// TwinCAT 3 PLC project UdpComm
// ProgramVersion: 3.1.4020.10
// libraries:
//   Tc2_Standard, * (Beckhoff Automation GmbH)
//   Tc2_System, * (Beckhoff Automation GmbH)
//   Tc2_Utilities, * (Beckhoff Automation GmbH)
//   Tc3_Interfaces, * (Beckhoff Automation GmbH)
//   Tc3_Module, * (Beckhoff Automation GmbH)
// project tree:
//   DUTs/ ModeStewart.TcDUT, RxRemote.TcDUT, ControlComau.TcDUT, RxComau.TcDUT, TxComau.TcDUT, RxMru.TcDUT, ControlStewart.TcDUT, TxRemote.TcDUT, FeedbackLeica.TcDUT, FeedbackComau.TcDUT, FeedbackMru.TcDUT, FeedbackStewart.TcDUT, TxHmi.TcDUT, TxHmiComau.TcDUT, TxHmiLeica.TcDUT, TxHmiMru.TcDUT, TxHmiStewart.TcDUT, TxStewart.TcDUT, RxStewart.TcDUT
//   / GlobalTextList.TcGTLO, TaskMAIN.TcTTO, Visualization Manager.TcVMO (not stored)
//   POUs/Kinematics/ EulerToBody.TcPOU, StewartTransform.TcPOU, xyz2zyx.TcPOU, zyx2xyz.TcPOU
//   POUs/LabEquipment/ LeicaInterface.TcPOU, RemoteInterface.TcPOU, MruInterface.TcPOU, ComauInterface.TcPOU, StewartInterface.TcPOU
//   POUs/ MAIN.TcPOU
//   POUs/Ship Simulation/ ShipSimulator.TcPOU, StocWave.TcPOU
//   POUs/UdpFBs/ FB_UdpClient.TcPOU (not stored), FB_UdpServer.TcPOU
// real-time tasks:
//   TASK TaskMAIN: cycle T#5ms, priority 20, ADS port 350
// I/O:
//   DEVICE EM1500 (RT-Ethernet Adapter)
//   DEVICE EM8000 (RT-Ethernet Adapter)
//   DEVICE COMAU (RT-Ethernet Adapter)
//   DEVICE REMOTE (RT-Ethernet Adapter)
//   DEVICE MRU2 (RT-Ethernet Adapter)
//   DEVICE MRU1 (RT-Ethernet Adapter)
//   DEVICE LeicaAT960 (EtherCAT), AmsNetId 169.254.76.98.11.1
//     Box 1 (Leica-RT-Output) [Leica RT Output]
// variable links:
//   UdpComm/UdpComm Instance <-> LeicaAT960 (EtherCAT)/Box 1 (Leica-RT-Output)
//     TaskMAIN Inputs/MAIN.at960.AngleHz <-> Cyclic Measurements/AngleHz
//     TaskMAIN Inputs/MAIN.at960.AngleVt <-> Cyclic Measurements/AngleVt
//     TaskMAIN Inputs/MAIN.at960.Distance <-> Cyclic Measurements/Distance
//     TaskMAIN Inputs/MAIN.at960.Quaternion{0..3} <-> Cyclic Measurements/Quaternion{0..3}  (4 links)
//     TaskMAIN Inputs/MAIN.at960.TimeStamp <-> Cyclic Measurements/TimeStamp

CONFIGURATION UdpComm
    RESOURCE PLC ON TwinCAT3
        TASK TaskMAIN(INTERVAL := T#5ms, PRIORITY := 20);
        PROGRAM MAIN WITH TaskMAIN : MAIN;
    END_RESOURCE
END_CONFIGURATION

// ---- DUTs/ModeStewart.TcDUT

TYPE ModeStewart :
(
	MODE_IDLE := 0,
	MODE_SIMULATOR,
	MODE_REMOTE,
	MODE_TRANSITION,
	MODE_GENERATOR,
	MODE_STOP
);
END_TYPE

// ---- DUTs/RxRemote.TcDUT
TYPE RxRemote :
STRUCT
	udp_key : DINT;
	comau : ControlComau;
END_STRUCT
END_TYPE

// ---- DUTs/ControlComau.TcDUT
TYPE ControlComau :
STRUCT
	q1 : REAL;
	q2 : REAL;
	q3 : REAL;
	q4 : REAL;
	q5 : REAL;
	q6 : REAL;
	q1_t : REAL;
	q2_t : REAL;
	q3_t : REAL;
	q4_t : REAL;
	q5_t : REAL;
	q6_t : REAL;
	q1_tt : REAL;
	q2_tt : REAL;
	q3_tt : REAL;
	q4_tt : REAL;
	q5_tt : REAL;
	q6_tt : REAL;
END_STRUCT
END_TYPE

// ---- DUTs/RxComau.TcDUT
TYPE RxComau :
STRUCT
	modalityActive : DINT;
	q1_ref : REAL;
	q2_ref : REAL;
	q3_ref : REAL;
	q4_ref : REAL;
	q5_ref : REAL; 
	q6_ref : REAL;
	q1 : REAL;
	q2 : REAL;
	q3 : REAL;
	q4 : REAL;
	q5 : REAL; 
	q6 : REAL;
	q1_t : REAL;
	q2_t : REAL;
	q3_t : REAL;
	q4_t : REAL;
	q5_t : REAL;
	q6_t : REAL;
	q1_tt : REAL;
	q2_tt : REAL;
	q3_tt : REAL;
	q4_tt : REAL;
	q5_tt : REAL;
	q6_tt : REAL;
END_STRUCT
END_TYPE

// ---- DUTs/TxComau.TcDUT
TYPE TxComau :
STRUCT
	udp_key	: DINT := 0;
	cmnd : DINT := 0;
	omega : REAL := 1.0;
	beta : REAL := 1.0;
	q1 : REAL := 0.0;
	q2 : REAL := 0.0;
	q3 : REAL := -90.0;
	q4 : REAL := 0.0;
	q5 : REAL := 90.0;
	q6 : REAL := 0.0;
	q1_t : REAL := 0.0;
	q2_t : REAL := 0.0;
	q3_t : REAL := 0.0;
	q4_t : REAL := 0.0;
	q5_t : REAL := 0.0;
	q6_t : REAL := 0.0;
	q1_tt : REAL := 0.0;
	q2_tt : REAL := 0.0;
	q3_tt : REAL := 0.0;
	q4_tt : REAL := 0.0;
	q5_tt : REAL := 0.0;
	q6_tt : REAL := 0.0;
END_STRUCT
END_TYPE

// ---- DUTs/RxMru.TcDUT
{attribute 'pack_mode' := '1'}
TYPE RxMru :
STRUCT
	mruOK : BYTE;
	dataLength : BYTE;
	token : BYTE;
	Temperature : REAL;
	PosMru_D : REAL;
	VelMru_D : REAL;
	AccMru_D : REAL;
	AngRate_D : REAL;
	Roll : REAL;
	Pitch : REAL;
	Yaw	: REAL;
	AngRate_R : REAL;
	AngRate_P : REAL;
	AngRate_Y : REAL;
	AngAcc_R : REAL;
	AngAcc_P : REAL;
	AngAcc_Y : REAL;
	VelMru_R : REAL;
	VelMru_P : REAL;
	VelMru_Y : REAL;
	AccMru_R : REAL;
	AccMru_P : REAL;
	AccMru_Y : REAL;
	checksum : BYTE;
END_STRUCT
END_TYPE

// ---- DUTs/ControlStewart.TcDUT
TYPE ControlStewart :
STRUCT
	surge : REAL := 0.0;
	sway : REAL := 0.0;
	heave : REAL := 0.0;
	phi : REAL := 0.0;
	theta : REAL := 0.0;
	psi : REAL := 0.0;
END_STRUCT
END_TYPE

// ---- DUTs/TxRemote.TcDUT
TYPE TxRemote :
STRUCT
	t : REAL := 0.0;
	em8000 : FeedbackStewart;	
	em1500 : FeedbackStewart;
	comau : FeedbackComau;
	at960 : FeedbackLeica;
	mru1 : FeedbackMru;
	mru2 : FeedbackMru;
END_STRUCT
END_TYPE

// ---- DUTs/FeedbackLeica.TcDUT
TYPE FeedbackLeica :
STRUCT
	x : REAL;
	y : REAL;
	z : REAL;
	q0 : REAL;
	q1 : REAL;
	q2 : REAL;
	q3 : REAL;
END_STRUCT
END_TYPE

// ---- DUTs/FeedbackComau.TcDUT
TYPE FeedbackComau :
STRUCT
	q1 : REAL;
	q2 : REAL;
	q3 : REAL;
	q4 : REAL;
	q5 : REAL;
	q6 : REAL;
	q1_t : REAL;
	q2_t : REAL;
	q3_t : REAL;
	q4_t : REAL;
	q5_t : REAL;
	q6_t : REAL;
	q1_tt : REAL;
	q2_tt : REAL;
	q3_tt : REAL;
	q4_tt : REAL;
	q5_tt : REAL;
	q6_tt : REAL;
END_STRUCT
END_TYPE

// ---- DUTs/FeedbackMru.TcDUT
TYPE FeedbackMru :
STRUCT
	heave : REAL;
	heave_t : REAL;
	heave_tt : REAL;
	turn_rate : REAL;
	roll : REAL;
	pitch : REAL;
	yaw : REAL;
	wx : REAL;
	wy : REAL;
	wz : REAL;
	wx_t : REAL;
	wy_t : REAL;
	wz_t : REAL;
	x_t : REAL;
	y_t : REAL;
	z_t : REAL;
	x_tt : REAL;
	y_tt : REAL;
	z_tt : REAL;
END_STRUCT
END_TYPE

// ---- DUTs/FeedbackStewart.TcDUT
TYPE FeedbackStewart :
STRUCT
	surge : REAL;
	sway : REAL;
	heave : REAL;
	phi : REAL;
	theta : REAL;
	psi	: REAL;
	surge_t	: REAL;
	sway_t	: REAL;
	heave_t	: REAL;
	wx : REAL;
	wy : REAL;
	wz : REAL;
	surge_tt : REAL;
	sway_tt : REAL;
	heave_tt : REAL;
	wx_t : REAL;
	wy_t : REAL;
	wz_t : REAL;
END_STRUCT
END_TYPE

// ---- DUTs/TxHmi.TcDUT
TYPE TxHmi :
STRUCT
	t : REAL := 0.0;
	em1500 : TxHmiStewart;
	em8000 : TxHmiStewart;
	comau : TxHmiComau;
	at960 : TxHmiLeica;	
	mru1 : TxHmiMru;
	mru2 : TxHmiMru;
END_STRUCT
END_TYPE

// ---- DUTs/TxHmiComau.TcDUT
TYPE TxHmiComau :
STRUCT
	status : DINT;
	q1 : REAL;
	q2 : REAL;
	q3 : REAL;
	q4 : REAL;
	q5 : REAL;
	q6 : REAL;
END_STRUCT
END_TYPE

// ---- DUTs/TxHmiLeica.TcDUT
TYPE TxHmiLeica :
STRUCT
	status : DINT;
	x : REAL;
	y : REAL;
	z : REAL;
	q0 : REAL;
	q1 : REAL;
	q2 : REAL;
	q3 : REAL;
END_STRUCT
END_TYPE

// ---- DUTs/TxHmiMru.TcDUT
TYPE TxHmiMru :
STRUCT
	status : DINT;
END_STRUCT
END_TYPE

// ---- DUTs/TxHmiStewart.TcDUT
TYPE TxHmiStewart :
STRUCT
	status : DINT;
	surge : REAL;
	sway : REAL;
	heave : REAL;
	phi : REAL;
	theta : REAL;
	psi	: REAL;
	surge_ref : REAL;
	sway_ref : REAL;
	heave_ref : REAL;
	phi_ref : REAL;
	theta_ref : REAL;
	psi_ref	: REAL;
	L1 : REAL;
	L2 : REAL;
	L3 : REAL;
	L4 : REAL;
	L5 : REAL;
	L6 : REAL;
	surge_sim : REAL;
	sway_sim : REAL;
	heave_sim : REAL;
	phi_sim : REAL;
	theta_sim : REAL;
	psi_sim	: REAL;
END_STRUCT
END_TYPE

// ---- DUTs/TxStewart.TcDUT
TYPE TxStewart :
STRUCT
	COUNT : DINT := 0;
	CMND : DINT := 0;
	AX : REAL := 0.0;
	AY : REAL := 0.0;
	AZ : REAL := 0.0;
	Dax : REAL := 0.0;
	Day : REAL := 0.0;
	Daz : REAL := 0.0;
	P_dot_CG : REAL := 0.0;
	Q_dot_CG : REAL := 0.0;
	R_dot_CG : REAL := 0.0;
	P_CG : REAL := 0.0;
	Q_CG : REAL := 0.0;
	R_CG : REAL := 0.0;
	Phi : REAL := 0.0;
	Theta : REAL := 0.0;
	U : REAL := 0.0;
	X_DIRECT : REAL := 0.0;
	Y_DIRECT : REAL := 0.0;
	Z_DIRECT : REAL := 0.0;
	X_CG : REAL := 0.0;
	Y_CG : REAL := 0.0;
	Z_CG : REAL := 0.0;
	Flags : REAL := 0.0;
	Bump_1 : REAL := 0.0;
	Bump_2 : REAL := 0.0;
	Bump_3 : REAL := 0.0;
	Bump_4 : REAL := 0.0;
	Bump_5 : REAL := 0.0;
	FREQ1 : REAL := 0.0;
	FREQ2 : REAL := 0.0;
	FREQ3 : REAL := 0.0;
	FREQ4 : REAL := 0.0;
	FREQ5 : REAL := 0.0;
	FREQ6 : REAL := 0.0;
	FREQ7 : REAL := 0.0;
	FREQ8 : REAL := 0.0;
	FREQ9 : REAL := 0.0;
	FREQ10 : REAL := 0.0;
	FREQ11 : REAL := 0.0;
	FREQ12 : REAL := 0.0;
	FREQ13 : REAL := 0.0;
	FREQ14 : REAL := 0.0;
	FREQ15 : REAL := 0.0;
	FREQ16 : REAL := 0.0;
	FREQ17 : REAL := 0.0;
	FREQ18 : REAL := 0.0;
	FREQ19 : REAL := 0.0;
	FREQ20 : REAL := 0.0;
	XGAIN1 : REAL := 0.0;
	XGAIN2 : REAL := 0.0;
	XGAIN3 : REAL := 0.0;
	XGAIN4 : REAL := 0.0;
	XGAIN5 : REAL := 0.0;
	XGAIN6 : REAL := 0.0;
	XGAIN7 : REAL := 0.0;
	XGAIN8 : REAL := 0.0;
	XGAIN9 : REAL := 0.0;
	XGAIN10 : REAL := 0.0;
	XGAIN11 : REAL := 0.0;
	XGAIN12 : REAL := 0.0;
	XGAIN13 : REAL := 0.0;
	XGAIN14 : REAL := 0.0;
	XGAIN15 : REAL := 0.0;
	XGAIN16 : REAL := 0.0;
	XGAIN17 : REAL := 0.0;
	XGAIN18 : REAL := 0.0;
	XGAIN19 : REAL := 0.0;
	XGAIN20 : REAL := 0.0;
	YGAIN1 : REAL := 0.0;
	YGAIN2 : REAL := 0.0;
	YGAIN3 : REAL := 0.0;
	YGAIN4 : REAL := 0.0;
	YGAIN5 : REAL := 0.0;
	YGAIN6 : REAL := 0.0;
	YGAIN7 : REAL := 0.0;
	YGAIN8 : REAL := 0.0;
	YGAIN9 : REAL := 0.0;
	YGAIN10 : REAL := 0.0;
	YGAIN11 : REAL := 0.0;
	YGAIN12 : REAL := 0.0;
	YGAIN13 : REAL := 0.0;
	YGAIN14 : REAL := 0.0;
	YGAIN15 : REAL := 0.0;
	YGAIN16 : REAL := 0.0;
	YGAIN17 : REAL := 0.0;
	YGAIN18 : REAL := 0.0;
	YGAIN19 : REAL := 0.0;
	YGAIN20 : REAL := 0.0;
	ZGAIN1 : REAL := 0.0;
	ZGAIN2 : REAL := 0.0;
	ZGAIN3 : REAL := 0.0;
	ZGAIN4 : REAL := 0.0;
	ZGAIN5 : REAL := 0.0;
	ZGAIN6 : REAL := 0.0;
	ZGAIN7 : REAL := 0.0;
	ZGAIN8 : REAL := 0.0;
	ZGAIN9 : REAL := 0.0;
	ZGAIN10 : REAL := 0.0;
	ZGAIN11 : REAL := 0.0;
	ZGAIN12 : REAL := 0.0;
	ZGAIN13 : REAL := 0.0;
	ZGAIN14 : REAL := 0.0;
	ZGAIN15 : REAL := 0.0;
	ZGAIN16 : REAL := 0.0;
	ZGAIN17 : REAL := 0.0;
	ZGAIN18 : REAL := 0.0;
	ZGAIN19 : REAL := 0.0;
	ZGAIN20 : REAL := 0.0;
	X_EXTRA : REAL := 0.0;
	Y_EXTRA : REAL := 0.0;
	Z_EXTRA : REAL := 0.0;
	PHI_EXTRA : REAL := 0.0;
	THETA_EXTRA : REAL := 0.0;
	PSI_EXTRA : REAL := 0.0;
	X_EXTRA_DOT : REAL := 0.0;
	Y_EXTRA_DOT : REAL := 0.0;
	Z_EXTRA_DOT : REAL := 0.0;
	PHI_EXTRA_DOT : REAL := 0.0;
	THETA_EXTRA_DOT : REAL := 0.0;
	PSI_EXTRA_DOT : REAL := 0.0;
	X_EXTRA_DDOT : REAL := 0.0;
	Y_EXTRA_DDOT : REAL := 0.0;
	Z_EXTRA_DDOT : REAL := 0.0;
	PHI_EXTRA_DDOT : REAL := 0.0;
	THETA_EXTRA_DDOT : REAL := 0.0;
	PSI_EXTRA_DDOT : REAL := 0.0;
END_STRUCT
END_TYPE

// ---- DUTs/RxStewart.TcDUT
TYPE RxStewart :
STRUCT
	Frame_Count : DINT := 0;
	Motion_Status : DINT := 0;
	Platform_setpoint_surge : REAL := 0.0;
	Platform_setpoint_sway : REAL := 0.0;
	Platform_setpoint_heave : REAL := 0.0;
	Platform_setpoint_roll : REAL := 0.0;
	Platform_setpoint_pitch : REAL := 0.0;
	Platform_setpoint_yaw : REAL := 0.0;
	Special_effect_surge_setpoint : REAL := 0.0;
	Special_effect_sway_setpoint : REAL := 0.0;
	Special_effect_heave_setpoint : REAL := 0.0;
	Special_effect_roll_setpoint : REAL := 0.0;
	Special_effect_pitch_setpoint : REAL := 0.0;
	Special_effect_yaw_setpoint : REAL := 0.0;
	Actual_position_actuator_1 : REAL := 0.0;
	Actual_position_actuator_2 : REAL := 0.0;
	Actual_position_actuator_3 : REAL := 0.0;
	Actual_position_actuator_4 : REAL := 0.0;
	Actual_position_actuator_5 : REAL := 0.0;
	Actual_position_actuator_6 : REAL := 0.0;
	Actual_platform_position_surge : REAL := 0.0;
	Actual_platform_position_sway : REAL := 0.0;
	Actual_platform_position_heave : REAL := 0.0;
	Actual_platform_position_roll : REAL := 0.0;
	Actual_platform_position_pitch : REAL := 0.0;
	Actual_platform_position_yaw : REAL := 0.0;
	Actual_platform_velocity_surge : REAL := 0.0;
	Actual_platform_velocity_sway : REAL := 0.0;
	Actual_platform_velocity_heave : REAL := 0.0;
	Actual_platform_velocity_roll : REAL := 0.0;
	Actual_platform_velocity_pitch : REAL := 0.0;
	Actual_platform_velocity_yaw : REAL := 0.0;
	Actual_platform_acceleration_surge : REAL := 0.0;
	Actual_platform_acceleration_sway : REAL := 0.0;
	Actual_platform_acceleration_heave : REAL := 0.0;
	Actual_platform_acceleration_roll : REAL := 0.0;
	Actual_platform_acceleration_pitch : REAL := 0.0;
	Actual_platform_acceleration_yaw : REAL := 0.0;
END_STRUCT
END_TYPE

// ---- POUs/MAIN.TcPOU
PROGRAM MAIN
VAR
	// HMI data
	hmi 				: TxHmi;	

	// Remote Interface	
	remote				: RemoteInterface(3232258620, 50060, 50050);
	
	// EtherCAT equipment
	at960				: LeicaInterface(ADR(hmi.at960));
	
	// UDP Equipment
	em1500				: StewartInterface(3232258591, 50031, 50041, 0, ADR(hmi.em1500));
	em8000				: StewartInterface(3232258590, 50030, 50040, 254, ADR(hmi.em8000));
	comau				: ComauInterface(3232258592, 50032, 50042, ADR(hmi.comau));
	
	mru1				: MruInterface(7551, ADR(hmi.mru1));
	mru2				: MruInterface(7552, ADR(hmi.mru2));
	
	
	counter				: UDINT := 0;
	
	
	
END_VAR

// Update remote data
remote();

// Update EtherCAT equipment
at960();

// Update UDP equipment
em1500();
em8000();
comau();
mru1();
mru2();

// Update timer
hmi.t := hmi.t + 5.0/1000.0;

END_PROGRAM

// ---- POUs/LabEquipment/RemoteInterface.TcPOU
{attribute 'c++_compatible'}
FUNCTION_BLOCK RemoteInterface IMPLEMENTS ITcIoUdpProtocolRecv
VAR_INPUT
	feedback			: TxRemote;
END_VAR
VAR_OUTPUT
	control 			: RxRemote;
END_VAR
VAR
	// UDP connection
	{attribute 'TcInitSymbol'}
	oid					: OTCID;
	ipUdp 				: ITcIoUdpProtocol;
	recvCounter			: UDINT := 0;
	sendCounter			: UDINT := 0;
	remoteUdpPort		: UINT;
	remoteIpAddr		: UDINT;	
	localUdpPort		: UINT;
	
	// UDP raw data
	rxUdpData			: RxRemote;
	txUdpData			: TxRemote;
	

END_VAR

VAR CONSTANT
	pi					: REAL := 3.141592653589793;
END_VAR


feedback.t := main.hmi.t;

// Update UDP data
UpdateUDP();

// Update IO data
UpdateIO();

METHOD FB_exit : BOOL
VAR_INPUT
	bInCopyCode : BOOL; // if TRUE, the exit method is called for exiting an instance that is copied afterwards (online change).
END_VAR
IF (NOT bInCopyCode AND ipUdp <> 0) THEN //Shutdown
	ipUdp.UnregisterReceiver(localUdpPort);
	FW_SafeRelease(ADR(ipUdp));
	FB_exit := TRUE;
ELSE
	FB_exit := FALSE;
END_IF
END_METHOD

METHOD FB_init : BOOL
VAR_INPUT
	bInitRetains 		: BOOL; // if TRUE, the retain variables are initialized (warm start / cold start)
	bInCopyCode 		: BOOL;  // if TRUE, the instance afterwards gets moved into the copy code (online change)
	
	_remoteIpAddr		: UDINT;
	_remoteUdpPort		: UINT;
	_localUdpPort		: UINT;
END_VAR

VAR
	ipSrv				: ITComObjectServer;
	hr 					: HRESULT;
END_VAR
// Initilize parameters
remoteIpAddr := _remoteIpAddr;
remoteUdpPort := _remoteUdpPort;
localUdpPort := _localUdpPort;

IF NOT bInCopyCode THEN // no online change
	IF ipUdp = 0 THEN
	    hr := FW_ObjMgr_GetObjectInstance(oid:=oid, iid:=TC_GLOBAL_IID_LIST.IID_ITcIoUdpProtocol, pipUnk:=ADR(ipUdp) );
		
		IF ( SUCCEEDED(hr) AND ipUdp.RegisterReceiver(localUdpPort, THIS^) = 0 ) THEN //open port
			FB_init := TRUE;
		ELSE
			FB_init := FALSE;			
			FW_SafeRelease(ADR(ipUdp));
		END_IF				
	END_IF
END_IF
END_METHOD

METHOD FB_reinit : BOOL
VAR_INPUT
END_VAR
IF (ipUdp <> 0) THEN 
  ipUdp.RegisterReceiver(localUdpPort, THIS^);
END_IF
END_METHOD

{attribute 'c++_compatible'}
{attribute 'signature_flag' := '33554688'}
{attribute 'pack_mode' := '4'}
{attribute 'show'}
{attribute 'minimal_input_size' := '4'}
{attribute 'checksuperglobal'}

METHOD ReceiveData : HRESULT
VAR_INPUT
	ipAddr	: UDINT;
	udpDestPort	: UINT;
	udpSrcPort	: UINT;
	nData	: UDINT;
	pData	: PVOID;
	pVlan	: POINTER TO ETYPE_VLAN_HEADER := 0;
END_VAR
IF (nData = SIZEOF(rxUdpData)) THEN
	// Copy recieved pData to rxUdpData
	MEMCPY(ADR(rxUdpData), pData, nData);
	
	// Count number of recieved UDP packets
	recvCounter := recvCounter + 1;
END_IF;
END_METHOD

{attribute 'c++_compatible'}
{attribute 'signature_flag' := '33554688'}
{attribute 'pack_mode' := '4'}
{attribute 'show'}
{attribute 'minimal_input_size' := '4'}
{attribute 'checksuperglobal'}

METHOD TcAddRef : UDINT
END_METHOD

{attribute 'c++_compatible'}
{attribute 'signature_flag' := '33554688'}
{attribute 'pack_mode' := '4'}
{attribute 'show'}
{attribute 'minimal_input_size' := '4'}
{attribute 'checksuperglobal'}

METHOD TcQueryInterface : HRESULT
VAR_INPUT
	iid	: REFERENCE TO IID;
	pipItf	: POINTER TO PVOID;
END_VAR
END_METHOD

{attribute 'c++_compatible'}
{attribute 'signature_flag' := '33554688'}
{attribute 'pack_mode' := '4'}
{attribute 'show'}
{attribute 'minimal_input_size' := '4'}
{attribute 'checksuperglobal'}

METHOD TcRelease : UDINT
END_METHOD

METHOD PRIVATE UpdateIO : BOOL
VAR_INPUT
END_VAR

control := rxUdpData;
txUdpData := feedback;
END_METHOD

METHOD PRIVATE UpdateUDP : BOOL
VAR_INPUT
END_VAR
// Send data to remote UDP server
IF ipUdp <> 0 THEN
	// Send data to remote UDP server
	ipUdp.SendData(remoteIpAddr, remoteUdpPort, localUdpPort, SIZEOF(txUdpData), ADR(txUdpData), TRUE, 0);
	sendCounter := sendCounter + 1;
	
	// Check for recieved data
	ipUdp.CheckReceived();
END_IF
END_METHOD

END_FUNCTION_BLOCK

// ---- POUs/LabEquipment/LeicaInterface.TcPOU
FUNCTION_BLOCK LeicaInterface
VAR_INPUT
END_VAR
VAR_OUTPUT
	feedback 			: FeedbackLeica;
END_VAR
VAR
	// Variables linked to LeicaAT960 Box 1
	AngleHz				AT %I* : LREAL := 0.0;
	AngleVt				AT %I* : LREAL := 0.0;
	Distance			AT %I* : LREAL := 0.0;
	Quaternion0			AT %I* : LREAL := 0.0;
	Quaternion1			AT %I* : LREAL := 0.0;
	Quaternion2			AT %I* : LREAL := 0.0;
	Quaternion3			AT %I* : LREAL := 0.0;
	TimeStamp			AT %I* : ULINT := 0;
	
	// Calculated cartesian positions
	x					: LREAL := 0.0;
	y					: LREAL := 0.0;
	z					: LREAL := 0.0;
	
	// HMI data
	pTxHmiData			: PVOID;
	txHmiData			: TxHmiLeica;
END_VAR

// Leica transform to x, y and z coordinates
x := Distance*SIN(AngleVt)*SIN(AngleHz);
y := Distance*SIN(AngleVt)*COS(AngleHz);
z := Distance*COS(AngleVt);

// Update IO data
UpdateIO();

// Update HMI data
UpdateHMI();

METHOD FB_init : BOOL
VAR_INPUT
	bInitRetains : BOOL; // if TRUE, the retain variables are initialized (warm start / cold start)
	bInCopyCode : BOOL;  // if TRUE, the instance afterwards gets moved into the copy code (online change)
	
	_pTxHmiData : PVOID;
END_VAR
pTxHmiData := _pTxHmiData;
END_METHOD

METHOD PRIVATE UpdateHMI : BOOL
VAR_INPUT
END_VAR
txHmiData.status := -1;

txHmiData.x := LREAL_TO_REAL(x);
txHmiData.y := LREAL_TO_REAL(y);
txHmiData.z := LREAL_TO_REAL(z);
txHmiData.q0 := LREAL_TO_REAL(Quaternion0);
txHmiData.q1 := LREAL_TO_REAL(Quaternion1);
txHmiData.q2 := LREAL_TO_REAL(Quaternion2);
txHmiData.q3 := LREAL_TO_REAL(Quaternion3);

// Update global HMI data
MEMCPY(pTxHmiData, ADR(txHmiData), SIZEOF(txHmiData));
END_METHOD

METHOD UpdateIO : BOOL
VAR_INPUT
END_VAR
// Update feedback data
feedback.x := LREAL_TO_REAL(x);
feedback.y := LREAL_TO_REAL(y);
feedback.z := LREAL_TO_REAL(z);
feedback.q0 := LREAL_TO_REAL(Quaternion0);
feedback.q1 := LREAL_TO_REAL(Quaternion1);
feedback.q2 := LREAL_TO_REAL(Quaternion2);
feedback.q3 := LREAL_TO_REAL(Quaternion3);
END_METHOD

END_FUNCTION_BLOCK

// ---- POUs/LabEquipment/StewartInterface.TcPOU
{attribute 'c++_compatible'}
FUNCTION_BLOCK StewartInterface IMPLEMENTS ITcIoUdpProtocolRecv
VAR_INPUT
	mode 				: ModeStewart;
	cmnd				: DINT := 0;
END_VAR
VAR_OUTPUT
	feedback 			: FeedbackStewart;
END_VAR
VAR
	// UDP connection
	{attribute 'TcInitSymbol'}
	oid					: OTCID;
	ipUdp 				: ITcIoUdpProtocol;
	recvCounter			: UDINT := 0;
	sendCounter			: UDINT := 0;
	remoteUdpPort		: UINT;
	remoteIpAddr		: UDINT;	
	localUdpPort		: UINT;
	
	// UDP raw data structures
	rxUdpData			: RxStewart;
	txUdpData			: TxStewart;
	
	// HMI data
	pTxHmiData			: PVOID;
	txHmiData			: TxHmiStewart;
	
	// Ship simulation
	seed				: INT;
	ship				: ShipSimulator(seed);

END_VAR

VAR CONSTANT
	pi					: REAL := 3.141592653589793;
END_VAR


// Update Ship simulation
ship();

// Update UDP data
UpdateUDP();

// Update IO data
UpdateIO();

// Update HMI data
UpdateHMI();

// State machine
mode := MODE_SIMULATOR;
CASE mode OF
	MODE_IDLE:
		//
	MODE_SIMULATOR:
		//
		txUdpData.CMND := cmnd;
		
		txUdpData.X_EXTRA := LREAL_TO_REAL(ship.surge);
		txUdpData.Y_EXTRA := LREAL_TO_REAL(ship.sway);
		txUdpData.Z_EXTRA := LREAL_TO_REAL(ship.heave);
		txUdpData.PHI_EXTRA := LREAL_TO_REAL(ship.phi);
		txUdpData.THETA_EXTRA := LREAL_TO_REAL(ship.theta);
		txUdpData.PSI_EXTRA := LREAL_TO_REAL(ship.psi);
		
	MODE_REMOTE:
		//
	MODE_TRANSITION:
		//
	MODE_GENERATOR:
		//
	MODE_STOP:
		//	
END_CASE

METHOD FB_exit : BOOL
VAR_INPUT
	bInCopyCode : BOOL; // if TRUE, the exit method is called for exiting an instance that is copied afterwards (online change).
END_VAR
IF (NOT bInCopyCode AND ipUdp <> 0) THEN //Shutdown
	ipUdp.UnregisterReceiver(localUdpPort);
	FW_SafeRelease(ADR(ipUdp));
	FB_exit := TRUE;
ELSE
	FB_exit := FALSE;
END_IF
END_METHOD

METHOD FB_init : BOOL
VAR_INPUT
	bInitRetains 		: BOOL; // if TRUE, the retain variables are initialized (warm start / cold start)
	bInCopyCode 		: BOOL;  // if TRUE, the instance afterwards gets moved into the copy code (online change)
	
	_remoteIpAddr		: UDINT;
	_remoteUdpPort		: UINT;
	_localUdpPort		: UINT;
	_seed				: INT;
	_pTxHmiData			: PVOID;
END_VAR

VAR
	ipSrv				: ITComObjectServer;
	hr 					: HRESULT;
END_VAR
// Initilize parameters
remoteIpAddr := _remoteIpAddr;
remoteUdpPort := _remoteUdpPort;
localUdpPort := _localUdpPort;
seed := _seed;
pTxHmiData :=_pTxHmiData;

IF NOT bInCopyCode THEN // no online change
	IF ipUdp = 0 THEN
	    hr := FW_ObjMgr_GetObjectInstance(oid:=oid, iid:=TC_GLOBAL_IID_LIST.IID_ITcIoUdpProtocol, pipUnk:=ADR(ipUdp) );
		
		IF ( SUCCEEDED(hr) AND ipUdp.RegisterReceiver(localUdpPort, THIS^) = 0 ) THEN //open port
			FB_init := TRUE;
		ELSE
			FB_init := FALSE;			
			FW_SafeRelease(ADR(ipUdp));
		END_IF				
	END_IF
END_IF
END_METHOD

METHOD FB_reinit : BOOL
VAR_INPUT
END_VAR
IF (ipUdp <> 0) THEN 
  ipUdp.RegisterReceiver(localUdpPort, THIS^);
END_IF
END_METHOD

{attribute 'c++_compatible'}
{attribute 'signature_flag' := '33554688'}
{attribute 'pack_mode' := '4'}
{attribute 'show'}
{attribute 'minimal_input_size' := '4'}
{attribute 'checksuperglobal'}

METHOD ReceiveData : HRESULT
VAR_INPUT
	ipAddr	: UDINT;
	udpDestPort	: UINT;
	udpSrcPort	: UINT;
	nData	: UDINT;
	pData	: PVOID;
	pVlan	: POINTER TO ETYPE_VLAN_HEADER := 0;
END_VAR
IF (nData = SIZEOF(rxUdpData)) THEN
	// Copy recieved pData to rxUdpData
	MEMCPY(ADR(rxUdpData), pData, nData);
	
	// Count number of recieved UDP packets
	recvCounter := recvCounter + 1;
END_IF;
END_METHOD

{attribute 'c++_compatible'}
{attribute 'signature_flag' := '33554688'}
{attribute 'pack_mode' := '4'}
{attribute 'show'}
{attribute 'minimal_input_size' := '4'}
{attribute 'checksuperglobal'}

METHOD TcAddRef : UDINT
END_METHOD

{attribute 'c++_compatible'}
{attribute 'signature_flag' := '33554688'}
{attribute 'pack_mode' := '4'}
{attribute 'show'}
{attribute 'minimal_input_size' := '4'}
{attribute 'checksuperglobal'}

METHOD TcQueryInterface : HRESULT
VAR_INPUT
	iid	: REFERENCE TO IID;
	pipItf	: POINTER TO PVOID;
END_VAR
END_METHOD

{attribute 'c++_compatible'}
{attribute 'signature_flag' := '33554688'}
{attribute 'pack_mode' := '4'}
{attribute 'show'}
{attribute 'minimal_input_size' := '4'}
{attribute 'checksuperglobal'}

METHOD TcRelease : UDINT
END_METHOD

METHOD PRIVATE UpdateHMI : BOOL
VAR_INPUT
END_VAR
// Updata HMI data
txHmiData.status := -1;

txHmiData.surge := rxUdpData.Actual_platform_position_surge;
txHmiData.sway := rxUdpData.Actual_platform_position_sway;
txHmiData.heave := rxUdpData.Actual_platform_position_heave;
txHmiData.phi := rxUdpData.Actual_platform_position_roll;
txHmiData.theta := rxUdpData.Actual_platform_position_pitch;
txHmiData.psi := rxUdpData.Actual_platform_position_yaw;

txHmiData.surge_ref := rxUdpData.Platform_setpoint_surge;
txHmiData.sway_ref := rxUdpData.Platform_setpoint_sway;
txHmiData.heave_ref := rxUdpData.Platform_setpoint_heave;
txHmiData.phi_ref := rxUdpData.Platform_setpoint_roll;
txHmiData.theta_ref := rxUdpData.Platform_setpoint_pitch;
txHmiData.psi_ref := rxUdpData.Platform_setpoint_yaw;

txHmiData.L1 := rxUdpData.Actual_position_actuator_1;
txHmiData.L2 := rxUdpData.Actual_position_actuator_2;
txHmiData.L3 := rxUdpData.Actual_position_actuator_3;
txHmiData.L4 := rxUdpData.Actual_position_actuator_4;
txHmiData.L5 := rxUdpData.Actual_position_actuator_5;
txHmiData.L6 := rxUdpData.Actual_position_actuator_6;

// Copy data to global HMI struct
MEMCPY(pTxHmidata, ADR(txHmiData), SIZEOF(TxHmiData));
END_METHOD

METHOD PRIVATE UpdateIO : BOOL
VAR_INPUT
END_VAR
// Update feedback data
feedback.surge 			:= rxUdpData.Actual_platform_position_surge;
feedback.sway 			:= rxUdpData.Actual_platform_position_sway;
feedback.heave 			:= rxUdpData.Actual_platform_position_heave;
feedback.phi 			:= rxUdpData.Actual_platform_position_roll;
feedback.theta 			:= rxUdpData.Actual_platform_position_pitch;
feedback.phi 			:= rxUdpData.Actual_platform_position_yaw;

feedback.surge_t		:= rxUdpData.Actual_platform_velocity_surge;
feedback.sway_t			:= rxUdpData.Actual_platform_velocity_sway;
feedback.heave_t		:= rxUdpData.Actual_platform_velocity_heave;
feedback.wx				:= rxUdpData.Actual_platform_velocity_roll;
feedback.wy				:= rxUdpData.Actual_platform_velocity_pitch;
feedback.wz				:= rxUdpData.Actual_platform_velocity_yaw;

feedback.surge_tt		:= rxUdpData.Actual_platform_acceleration_surge;
feedback.sway_tt		:= rxUdpData.Actual_platform_acceleration_sway;
feedback.heave_tt		:= rxUdpData.Actual_platform_acceleration_heave;
feedback.wx_t			:= rxUdpData.Actual_platform_acceleration_roll;
feedback.wy_t			:= rxUdpData.Actual_platform_acceleration_pitch;
feedback.wz_t			:= rxUdpData.Actual_platform_acceleration_yaw;
END_METHOD

METHOD PRIVATE UpdateUDP : BOOL
VAR_INPUT
END_VAR
// Send data to remote UDP server
IF ipUdp <> 0 THEN
	// Send data to remote UDP server
	ipUdp.SendData(remoteIpAddr, remoteUdpPort, localUdpPort, SIZEOF(txUdpData), ADR(txUdpData), TRUE, 0);
	sendCounter := sendCounter + 1;
	
	// Check for recieved data
	ipUdp.CheckReceived();
END_IF

// Update counter
txUdpData.COUNT 		:= txUdpData.COUNT + 1;
END_METHOD

METHOD PRIVATE xyz2zyx : ARRAY [0..2] OF REAL
VAR_INPUT
	phi : ARRAY [0..2] OF REAL;
END_VAR

VAR
	t1: REAL;
	t2: REAL;
	t3: REAL;
	t4: REAL;
	t5: REAL;
	t6: REAL;
	t7: REAL;
	t8: REAL;
END_VAR
// Maple optimized code
t1 := COS(phi[0]);
t2 := SIN(phi[1]);
t3 := SIN(phi[2]);
t4 := SIN(phi[0]);
t5 := COS(phi[2]);
t6 := t1 * t3;
t7 := t4 * t5;
t8 := COS(phi[1]);

xyz2zyx[0] := ATAN((t6 * t2 + t7)/(t1 * t8));
xyz2zyx[1] := -ASIN(-t1 * t2 * t5 + t3 * t4);
xyz2zyx[2] := ATAN((t7 * t2 + t6)/(t5 * t8));
END_METHOD

METHOD PRIVATE zyx2xyz : ARRAY [0..2] OF REAL
VAR_INPUT
	phi : ARRAY [0..2] OF REAL;
END_VAR

VAR
	t1: REAL;
	t2: REAL;
	t3: REAL;
	t4: REAL;
	t5: REAL;
	t6: REAL;
	t7: REAL;
	t8: REAL;
END_VAR
// Maple optimized code
t1 := SIN(phi[0]);
t2 := COS(phi[2]);
t3 := COS(phi[0]);
t4 := SIN(phi[1]);
t5 := SIN(phi[2]);
t6 := t3 * t5;
t7 := t1 * t2;
t8 := COS(phi[1]);

zyx2xyz[0] := ATAN((-t6 * t4 + t7)/(t3 * t8));
zyx2xyz[1] := ASIN(t3 * t4 * t2 + t1 * t5);
zyx2xyz[2] := ATAN((-t7 * t4 + t6)/( t2 * t8));
END_METHOD

END_FUNCTION_BLOCK

// ---- POUs/Ship Simulation/ShipSimulator.TcPOU
FUNCTION_BLOCK ShipSimulator
VAR_INPUT
	timestep : LREAL := 0.005;
	
	// Default wavespectrum(Hs=8.0, T1=12.0, spec='JONSWAP')
    w0 : LREAL :=  0.43567172549;
    lambda : LREAL :=  0.101904641875;
    sigma : LREAL :=  5.3310138243;
	
	// PD Contoroller poles
	poles : LREAL := 0.3;
	
	// Max output states allowed
	surge_max : LREAL := 0.2;
	sway_max : LREAL := 0.2;
	heave_max : LREAL := 0.4;
	phi_max : LREAL := 5.0/180.0*pi;
	theta_max : LREAL := 5.0/180.0*pi;
	psi_max : LREAL := 5.0/180.0*pi;
	
	
END_VAR
VAR_OUTPUT
	t : LREAL := 0.0;
	
	surge : LREAL;
	sway : LREAL;
	heave : LREAL;
	phi : LREAL;
	theta : LREAL;
	psi : LREAL;
END_VAR
VAR
	// Counter variable
	dof : UINT;
	
	// Random generator, initialized in FB_init
	rand : DRAND;

	//  Ship 1st order dynamics from system identification
	Ts_x : LREAL := 45.215;
    Ts_y : LREAL := 18.335;
    Ts_yaw : LREAL := 16.425;
    K_x : LREAL := 1.49944614059E-07;
    K_y : LREAL := 1.13435297558E-07;
    K_yaw : LREAL := 2.77309521498E-10;
	
	// State vectors
	states : ARRAY [0..23] OF LREAL;
	eta : ARRAY [0..5] OF LREAL;
	
	// Scaling gains
	eta_max : ARRAY [0..5] OF LREAL;
	Ks : ARRAY [0..5] OF LREAL := [1.0, 1.0, 1.0, 1.0, 1.0, 1.0];
END_VAR

// Integrate solution by one timestep
integrate();

// Red max settings
eta_max[0] := ABS(surge_max);
eta_max[1] := ABS(sway_max);
eta_max[2] := ABS(heave_max);
eta_max[3] := ABS(phi_max);
eta_max[4] := ABS(theta_max);
eta_max[5] := ABS(psi_max);

// Adapt output to fit defined maximum limits
FOR dof := 0 TO 5 DO
	IF ABS(Ks[dof]*states[dof]) >= ABS(eta_max[dof]) THEN
		IF ABS(states[dof]) <> 0.0 THEN
			Ks[dof] := eta_max[dof]/ABS(states[dof]);
		END_IF	
	END_IF	
END_FOR


surge := Ks[0]*states[0];
sway := Ks[1]*states[1];
heave := Ks[2]*states[2];
phi := Ks[3]*states[3];
theta := Ks[4]*states[4];
psi := Ks[5]*states[5];

METHOD FB_init : BOOL
VAR_INPUT
	bInitRetains : BOOL; // if TRUE, the retain variables are initialized (warm start / cold start)
	bInCopyCode : BOOL;  // if TRUE, the instance afterwards gets moved into the copy code (online change)
	
	seed : INT;
END_VAR
// Define seed number for stochastic wave
rand.Seed := seed;
END_METHOD

METHOD PRIVATE integrate : BOOL
VAR_INPUT
END_VAR

VAR
	i : DINT;
	
	states_t : ARRAY [0..23] OF LREAL;
END_VAR


states_t := ode(states);

FOR i := 0 TO 23 DO
	states[i] := states[i] + states_t[i]*timestep;
END_FOR

t := t + timestep;
END_METHOD

METHOD PRIVATE kinematics : ARRAY [0..5] OF LREAL;
VAR_INPUT
	eta : ARRAY [0..5] OF LREAL;
	v : ARRAY [0..5] OF LREAL;
END_VAR

VAR
	eta_t : ARRAY[0..5] OF LREAL;
END_VAR

IF COS(eta[4]) <> 0.0 THEN
	eta_t[0] := -v[1]*(COS(eta[3])*SIN(eta[5])-COS(eta[5])*SIN(eta[3])*SIN(eta[4]))+v[2]*(SIN(eta[3])*SIN(eta[5])+COS(eta[3])*COS(eta[5])*SIN(eta[4]))+v[0]*COS(eta[4])*COS(eta[5]);
	eta_t[1] := v[1]*(COS(eta[3])*COS(eta[5])+SIN(eta[3])*SIN(eta[4])*SIN(eta[5]))-v[2]*(COS(eta[5])*SIN(eta[3])-COS(eta[3])*SIN(eta[4])*SIN(eta[5]))+v[0]*COS(eta[4])*SIN(eta[5]);
	eta_t[2] := -v[0]*SIN(eta[4])+v[2]*COS(eta[3])*COS(eta[4])+v[1]*COS(eta[4])*SIN(eta[3]);
	eta_t[3] := v[3]+(v[5]*COS(eta[3])*SIN(eta[4]))/COS(eta[4])+(v[4]*SIN(eta[3])*SIN(eta[4]))/COS(eta[4]);
	eta_t[4] := v[4]*COS(eta[3])-v[5]*SIN(eta[3]);
	eta_t[5] := (v[5]*COS(eta[3]))/COS(eta[4])+(v[4]*SIN(eta[3]))/COS(eta[4]);
	
	kinematics := eta_t;
END_IF;
END_METHOD

METHOD PRIVATE ode : ARRAY [0..23] OF LREAL
VAR_INPUT
	y : ARRAY [0..23] OF LREAL;
END_VAR

VAR
	// Wave component gains
	K : ARRAY [0..5] OF LREAL := [1E4, 1E4, 4E8, 1E8, 1E5, 1E7];	
	
	// PD Controller gains
	Kp : LREAL;
	Kd : LREAL;	
	
	w : LREAL;
	i : UINT;
	
	eta : ARRAY [0..5] OF LREAL;
	eta_t : ARRAY [0..5] OF LREAL;
	
	v : ARRAY [0..5] OF LREAL;
	v_t : ARRAY [0..5] OF LREAL;
	
	x : ARRAY [0..11] OF LREAL;
	x_t : ARRAY [0..11] OF LREAL;
	
	tau : ARRAY [0..5] OF LREAL;
	tau_wave : ARRAY [0..5] OF LREAL;
	tau_tot : ARRAY [0..5] OF LREAL;

	y_t : ARRAY [0..23] OF LREAL;
END_VAR
// Rigid body states
FOR i := 0 TO 5 DO
	eta[i] := y[i];
	v[i] := y[i+6];
END_FOR; 

// Wave simulation states
FOR i := 0 TO 11 DO
	x[i] := y[i+12];
END_FOR

//*******************************************************************//

// Kinematics
eta_t := kinematics(eta, v);

// Wave forces driven by random process
FOR i := 0 TO 5 DO
	rand();
	w := rand.Num*2.0 - 1.0;
	
	x_t[0 + 2*i] := x[1 + 2*i];
	x_t[1 + 2*i] := 2*w*ABS(lambda*sigma*w0) - w0*w0*x[0 + 2*i] - 2*x[1 + 2*i]*ABS(lambda*w0);
	tau_wave[i] := ABS(K[i])*x[1 + 2*i];	
END_FOR;

// PD Controller for DP simulation in surge, sway and yaw directions
Kp := poles*poles*2.0/K_x;
Kd := (2.0*ABS(poles) - 4.0/Ts_x)/K_x;
tau[0] := -(Kp*eta[0] + Kd*eta_t[0]);

Kp := poles*poles*2.0/K_y;
Kd := (2.0*ABS(poles) - 4.0/Ts_y)/K_y;
tau[1] := -(Kp*eta[1] + Kd*eta_t[1]);

Kp := poles*poles*2.0/K_yaw;
Kd := (2.0*ABS(poles) - 4.0/Ts_yaw)/K_yaw;
tau[5] := -(Kp*eta[5] + Kd*eta_t[5]);


// Total forces
tau_tot[0] := tau[0] + tau_wave[0];
tau_tot[1] := tau[1] + tau_wave[1];
tau_tot[2] := tau[2] + tau_wave[2];
tau_tot[3] := tau[3] + tau_wave[3];
tau_tot[4] := tau[4] + tau_wave[4];
tau_tot[5] := tau[5] + tau_wave[5];

// Rigid ship ODE >> v_t = Minv*(-D*v - G*eta + tau + tau_wave)
v_t[0] := 0.000000146900537469*tau_tot[0] - 1.15779191741*eta[4] - 0.00633181020913*eta[2] - 0.000000000481800095922*tau_tot[2] + 0.000000000184278003677*tau_tot[4] - 0.0866236024535*v[0] - 0.00613744736768*v[2] - 0.274323279079*v[4];
v_t[1] := 0.55557891964*eta[3] + 0.000000132912419336*tau_tot[1] - 0.00000000415239105737*tau_tot[3] + 0.0000000000224611856126*tau_tot[5] - 0.253122582192*v[1] - 0.104731972248*v[3] - 0.980405576225*v[5];
v_t[2] := 0.0000000575501415202*tau_tot[2] - 1.50179843329*eta[4] - 0.000000000481800095922*tau_tot[0] - 0.772453112071*eta[2] - 0.000000000397149205293*tau_tot[4] + 0.000284105563467*v[0] - 0.0741429429368*v[2] - 1.51936619529*v[4];
v_t[3] := 0.00000000289648823017*tau_tot[3] - 0.00000000415239105737*tau_tot[1] - 0.387542449503*eta[3] + 0.000000000048718802883*tau_tot[5] + 0.00236474400079*v[1] - 0.0922339025763*v[3] + 0.117970498295*v[5];
v_t[4] := 0.000000000184278003677*tau_tot[0] - 0.954371208694*eta[4] - 0.00521932937313*eta[2] - 0.000000000397149205293*tau_tot[2] + 0.000000000151900888631*tau_tot[4] - 0.00010866416697*v[0] - 0.00505911552371*v[2] - 0.226125468221*v[4];
v_t[5] := 0.0000000000224611856126*tau_tot[1] - 0.00651844672092*eta[3] + 0.000000000048718802883*tau_tot[3] + 0.000000000280999799559*tau_tot[5] - 0.0017495572239*v[1] + 0.0115949285132*v[3] - 0.249188054934*v[5];



//*******************************************************************//

// Rigid body states
FOR i := 0 TO 5 DO
	y_t[i] := eta_t[i];
	y_t[i+6] := v_t[i];
END_FOR; 

// Wave simulation states
FOR i := 0 TO 11 DO
	y_t[i+12] := x_t[i];
END_FOR

// Return y_t
ode := y_t;
END_METHOD

END_FUNCTION_BLOCK

// ---- POUs/Kinematics/xyz2zyx.TcPOU
FUNCTION xyz2zyx : ARRAY [0..2] of REAL
VAR_INPUT
	phi : ARRAY [0..2] OF REAL;
END_VAR
VAR
	t1: REAL;
	t2: REAL;
	t3: REAL;
	t4: REAL;
	t5: REAL;
	t6: REAL;
	t7: REAL;
	t8: REAL;
END_VAR

// Maple optimized code
t1 := COS(phi[0]);
t2 := SIN(phi[1]);
t3 := SIN(phi[2]);
t4 := SIN(phi[0]);
t5 := COS(phi[2]);
t6 := t1 * t3;
t7 := t4 * t5;
t8 := COS(phi[1]);

xyz2zyx[0] := ATAN((t6 * t2 + t7)/(t1 * t8));
xyz2zyx[1] := -ASIN(-t1 * t2 * t5 + t3 * t4);
xyz2zyx[2] := ATAN((t7 * t2 + t6)/(t5 * t8));

END_FUNCTION

// ---- POUs/Kinematics/zyx2xyz.TcPOU
FUNCTION zyx2xyz : ARRAY [0..2] OF REAL
VAR_INPUT
	phi : ARRAY [0..2] of REAL;
END_VAR
VAR
	t1: REAL;
	t2: REAL;
	t3: REAL;
	t4: REAL;
	t5: REAL;
	t6: REAL;
	t7: REAL;
	t8: REAL;
END_VAR

// Maple optimized code
t1 := SIN(phi[0]);
t2 := COS(phi[2]);
t3 := COS(phi[0]);
t4 := SIN(phi[1]);
t5 := SIN(phi[2]);
t6 := t3 * t5;
t7 := t1 * t2;
t8 := COS(phi[1]);

zyx2xyz[0] := ATAN((-t6 * t4 + t7)/(t3 * t8));
zyx2xyz[1] := ASIN(t3 * t4 * t2 + t1 * t5);
zyx2xyz[2] := ATAN((-t7 * t4 + t6)/( t2 * t8));

END_FUNCTION

// ---- POUs/LabEquipment/ComauInterface.TcPOU
{attribute 'c++_compatible'}
FUNCTION_BLOCK ComauInterface IMPLEMENTS ITcIoUdpProtocolRecv
VAR_INPUT
	cmnd				: DINT;
	control				: ControlComau;
END_VAR
VAR_OUTPUT
	feedback			: FeedbackComau;
END_VAR
VAR
	// UDP connection
	{attribute 'TcInitSymbol'}
	oid					: OTCID;
	ipUdp 				: ITcIoUdpProtocol;
	recvCounter			: UDINT := 0;
	sendCounter			: UDINT := 0;
	remoteUdpPort		: UINT;
	remoteIpAddr		: UDINT;	
	localUdpPort		: UINT;
	
	// UDP raw data structures
	rxUdpData			: RxComau;
	txUdpData			: TxComau;
	
	// HMI data
	pTxHmiData			: PVOID;
	txHmiData			: TxHmiComau;
	
	
END_VAR


txUdpData.cmnd := cmnd;

// Update UDP data
UpdateUDP();

// Update IO data
UpdateIO();

// Update HMI data
UpdateHMI();

METHOD FB_exit : BOOL
VAR_INPUT
	bInCopyCode : BOOL; // if TRUE, the exit method is called for exiting an instance that is copied afterwards (online change).
END_VAR
IF (NOT bInCopyCode AND ipUdp <> 0) THEN //Shutdown
	ipUdp.UnregisterReceiver(localUdpPort);
	FW_SafeRelease(ADR(ipUdp));
	FB_exit := TRUE;
ELSE
	FB_exit := FALSE;
END_IF
END_METHOD

METHOD FB_init : BOOL
VAR_INPUT
	bInitRetains		: BOOL; // if TRUE, the retain variables are initialized (warm start / cold start)
	bInCopyCode			: BOOL;  // if TRUE, the instance afterwards gets moved into the copy code (online change)
	
	// Contructor arguments
	_remoteIpAddr		: UDINT;
	_remoteUdpPort 		: UINT;
	_localUdpPort	 	: UINT;
	_pTxHmiData			: PVOID;
END_VAR

VAR
	ipSrv				: ITComObjectServer;
	hr 					: HRESULT;
END_VAR
// Initilize parameters
remoteIpAddr := _remoteIpAddr;
remoteUdpPort := _remoteUdpPort;
localUdpPort := _localUdpPort;
pTxHmiData := _pTxHmiData;

IF NOT bInCopyCode THEN // no online change
	IF ipUdp = 0 THEN
	    hr := FW_ObjMgr_GetObjectInstance(oid:=oid, iid:=TC_GLOBAL_IID_LIST.IID_ITcIoUdpProtocol, pipUnk:=ADR(ipUdp) );
		
		IF ( SUCCEEDED(hr) AND ipUdp.RegisterReceiver(localUdpPort, THIS^) = 0 ) THEN //open port
			FB_init := TRUE;
		ELSE
			FB_init := FALSE;			
			FW_SafeRelease(ADR(ipUdp));
		END_IF				
	END_IF
END_IF
END_METHOD

METHOD FB_reinit : BOOL
VAR_INPUT
END_VAR
IF (ipUdp <> 0) THEN 
  ipUdp.RegisterReceiver(localUdpPort, THIS^);
END_IF
END_METHOD

{attribute 'c++_compatible'}
{attribute 'signature_flag' := '33554688'}
{attribute 'pack_mode' := '4'}
{attribute 'show'}
{attribute 'minimal_input_size' := '4'}
{attribute 'checksuperglobal'}

METHOD ReceiveData : HRESULT
VAR_INPUT
	ipAddr	: UDINT;
	udpDestPort	: UINT;
	udpSrcPort	: UINT;
	nData	: UDINT;
	pData	: PVOID;
	pVlan	: POINTER TO ETYPE_VLAN_HEADER := 0;
END_VAR
IF (nData = SIZEOF(rxUdpData)) THEN
	// Copy recieved pData to rxUdpData
	MEMCPY(ADR(rxUdpData), pData, nData);
	
	// Count number of recieved UDP packets
	recvCounter := recvCounter + 1;
END_IF;
END_METHOD

{attribute 'c++_compatible'}
{attribute 'signature_flag' := '33554688'}
{attribute 'pack_mode' := '4'}
{attribute 'show'}
{attribute 'minimal_input_size' := '4'}
{attribute 'checksuperglobal'}

METHOD TcAddRef : UDINT
END_METHOD

{attribute 'c++_compatible'}
{attribute 'signature_flag' := '33554688'}
{attribute 'pack_mode' := '4'}
{attribute 'show'}
{attribute 'minimal_input_size' := '4'}
{attribute 'checksuperglobal'}

METHOD TcQueryInterface : HRESULT
VAR_INPUT
	iid	: REFERENCE TO IID;
	pipItf	: POINTER TO PVOID;
END_VAR
END_METHOD

{attribute 'c++_compatible'}
{attribute 'signature_flag' := '33554688'}
{attribute 'pack_mode' := '4'}
{attribute 'show'}
{attribute 'minimal_input_size' := '4'}
{attribute 'checksuperglobal'}

METHOD TcRelease : UDINT
END_METHOD

METHOD PRIVATE UpdateHMI : BOOL
VAR_INPUT
END_VAR
txHmiData.status := -1;

txHmiData.q1 := rxUdpData.q1;
txHmiData.q2 := rxUdpData.q2;
txHmiData.q3 := rxUdpData.q3;
txHmiData.q4 := rxUdpData.q4;
txHmiData.q5 := rxUdpData.q5;
txHmiData.q6 := rxUdpData.q6;

// Update global HMI data
MEMCPY(pTxHmiData, ADR(txHmiData), SIZEOF(txHmiData));
END_METHOD

METHOD PRIVATE UpdateIO : BOOL
VAR_INPUT
END_VAR
// Control data
txUdpData.q1 := control.q1;
txUdpData.q2 := control.q2;
txUdpData.q3 := control.q3;
txUdpData.q4 := control.q4;
txUdpData.q5 := control.q5;
txUdpData.q6 := control.q6;
txUdpData.q1_t := control.q1_t;
txUdpData.q2_t := control.q2_t;
txUdpData.q3_t := control.q3_t;
txUdpData.q4_t := control.q4_t;
txUdpData.q5_t := control.q5_t;
txUdpData.q6_t := control.q6_t;
txUdpData.q1_tt := control.q1_tt;
txUdpData.q2_tt := control.q2_tt;
txUdpData.q3_tt := control.q3_tt;
txUdpData.q4_tt := control.q4_tt;
txUdpData.q5_tt := control.q5_tt;
txUdpData.q6_tt := control.q6_tt;

// Feedback data
feedback.q1 := rxUdpData.q1;
feedback.q2 := rxUdpData.q2;
feedback.q3 := rxUdpData.q3;
feedback.q4 := rxUdpData.q4;
feedback.q5 := rxUdpData.q5;
feedback.q6 := rxUdpData.q6;
feedback.q1_t := rxUdpData.q1_t;
feedback.q2_t := rxUdpData.q2_t;
feedback.q3_t := rxUdpData.q3_t;
feedback.q4_t := rxUdpData.q4_t;
feedback.q5_t := rxUdpData.q5_t;
feedback.q6_t := rxUdpData.q6_t;
feedback.q1_tt := rxUdpData.q1_tt;
feedback.q2_tt := rxUdpData.q2_tt;
feedback.q3_tt := rxUdpData.q3_tt;
feedback.q4_tt := rxUdpData.q4_tt;
feedback.q5_tt := rxUdpData.q5_tt;
feedback.q6_tt := rxUdpData.q6_tt;
END_METHOD

METHOD PRIVATE UpdateUDP : BOOL
VAR_INPUT
END_VAR
// Send data to remote UDP server
IF ipUdp <> 0 THEN
	// Send data to remote UDP server
	ipUdp.SendData(remoteIpAddr, remoteUdpPort, localUdpPort, SIZEOF(txUdpData), ADR(txUdpData), TRUE, 0);
	sendCounter := sendCounter + 1;
	
	// Check for recieved data
	ipUdp.CheckReceived();
END_IF

txUdpData.udp_key := 32;
txUdpData.cmnd := 0;
txUdpData.beta := 1.0;
txUdpData.omega := 1.0;
END_METHOD

END_FUNCTION_BLOCK

// ---- POUs/LabEquipment/MruInterface.TcPOU
{attribute 'c++_compatible'}
FUNCTION_BLOCK MruInterface IMPLEMENTS ITcIoUdpProtocolRecv
VAR_INPUT
	
END_VAR
VAR_OUTPUT
	feedback			: FeedbackMru;
END_VAR
VAR	
	// UDP connection
	{attribute 'TcInitSymbol'}
	oid					: OTCID;
	ipUdp 				: ITcIoUdpProtocol;
	recvCounter			: UDINT := 0;
	localUdpPort		: UINT;
	
	// UDP raw data structures
	rxUdpDataBE			: RxMru;	// Big endian data struct
	rxUdpData			: RxMru;	// Host/little endian data struct
	
	// HMI data
	pTxHmiData			: PVOID;
	txHmiData			: TxHmiMru;
END_VAR

// Update UDP data
UpdateUDP();

// Update IO data
UpdateIO();

// Update HMI data
UpdateHMI();

METHOD BigToLittleEndian : REAL
VAR_INPUT
	realIn		: REAL;
END_VAR

VAR
	realOut		: REAL;	

	bytesIn		: ARRAY [0..3] OF BYTE;
	bytesOut	: ARRAY [0..3] OF BYTE;
END_VAR
// Copy to byte array
MEMCPY(ADR(bytesIn), ADR(realIn), 4);

// Switch bytes
bytesOut[3] := bytesIn[0];
bytesOut[2] := bytesIn[1];
bytesOut[1] := bytesIn[2];
bytesOut[0] := bytesIn[3];

// Copy switched butes to realOut
MEMCPY(ADR(realOut), ADR(bytesOut), 4);

// Return switched version of realIn
BigToLittleEndian := realOut;
END_METHOD

METHOD FB_exit : BOOL
VAR_INPUT
	bInCopyCode : BOOL; // if TRUE, the exit method is called for exiting an instance that is copied afterwards (online change).
END_VAR
IF (NOT bInCopyCode AND ipUdp <> 0) THEN //Shutdown
	ipUdp.UnregisterReceiver(localUdpPort);
	FW_SafeRelease(ADR(ipUdp));
	FB_exit := TRUE;
ELSE
	FB_exit := FALSE;
END_IF
END_METHOD

METHOD FB_init : BOOL
VAR_INPUT
	bInitRetains 		: BOOL; // if TRUE, the retain variables are initialized (warm start / cold start)
	bInCopyCode 		: BOOL;  // if TRUE, the instance afterwards gets moved into the copy code (online change)
	
	// Contructor arguments
	_localUdpPort 		: UINT;
	_pTxHmiData			: PVOID;
END_VAR

VAR
	ipSrv				: ITComObjectServer;
	hr 					: HRESULT;
END_VAR
// Initilize parameters
localUdpPort := _localUdpPort;
pTxHmiData := _pTxHmiData;

IF NOT bInCopyCode THEN // no online change
	IF ipUdp = 0 THEN
	    hr := FW_ObjMgr_GetObjectInstance(oid:=oid, iid:=TC_GLOBAL_IID_LIST.IID_ITcIoUdpProtocol, pipUnk:=ADR(ipUdp) );
		
		IF (SUCCEEDED(hr) AND ipUdp.RegisterReceiver(localUdpPort, THIS^) = 0 ) THEN //open local port
			FB_init := TRUE;
		ELSE
			FB_init := FALSE;			
			FW_SafeRelease(ADR(ipUdp));
		END_IF				
	END_IF
END_IF
END_METHOD

METHOD FB_reinit : BOOL
VAR_INPUT
END_VAR
IF (ipUdp <> 0) THEN 
	ipUdp.RegisterReceiver(localUdpPort, THIS^);
END_IF
END_METHOD

{attribute 'c++_compatible'}
{attribute 'signature_flag' := '33554688'}
{attribute 'pack_mode' := '1'}
{attribute 'show'}
{attribute 'minimal_input_size' := '4'}
{attribute 'checksuperglobal'}
METHOD ReceiveData : HRESULT
VAR_INPUT
	ipAddr			: UDINT;
	udpDestPort		: UINT;
	udpSrcPort		: UINT;
	nData			: UDINT;
	pData			: PVOID;
	pVlan			: POINTER TO ETYPE_VLAN_HEADER := 0;
END_VAR
// Send and receive data if the received data size is correct
IF (nData = SIZEOF(RxMru)) THEN
	// Count number of recieved UDP packets
	recvCounter := recvCounter + 1;

	// Copy data to recv buffer
	MEMCPY(ADR(rxUdpDataBE), pData, nData);
END_IF
END_METHOD

{attribute 'c++_compatible'}
{attribute 'signature_flag' := '33554688'}
{attribute 'pack_mode' := '1'}
{attribute 'show'}
{attribute 'minimal_input_size' := '4'}
{attribute 'checksuperglobal'}
METHOD TcAddRef : UDINT
END_METHOD

{attribute 'c++_compatible'}
{attribute 'signature_flag' := '33554688'}
{attribute 'pack_mode' := '1'}
{attribute 'show'}
{attribute 'minimal_input_size' := '4'}
{attribute 'checksuperglobal'}
METHOD TcQueryInterface : HRESULT
VAR_INPUT
	iid	: REFERENCE TO IID;
	pipItf	: POINTER TO PVOID;
END_VAR
END_METHOD

{attribute 'c++_compatible'}
{attribute 'signature_flag' := '33554688'}
{attribute 'pack_mode' := '1'}
{attribute 'show'}
{attribute 'minimal_input_size' := '4'}
{attribute 'checksuperglobal'}
METHOD TcRelease : UDINT
END_METHOD

METHOD PRIVATE UpdateHMI : BOOL
VAR_INPUT
END_VAR
txHmiData.status := -1;


// Update global HMI data
MEMCPY(pTxHmiData, ADR(txHmiData), SIZEOF(txHmiData));
END_METHOD

METHOD PRIVATE UpdateIO : BOOL
VAR_INPUT
END_VAR
// Update feedback data
feedback.heave := rxUdpData.PosMru_D;
feedback.heave_t := rxUdpData.VelMru_D;
feedback.heave_tt := rxUdpData.AccMru_D;
feedback.turn_rate := rxUdpData.AngRate_D;
feedback.roll := rxUdpData.Roll;
feedback.pitch := rxUdpData.Pitch;
feedback.yaw := rxUdpData.Yaw;
feedback.wx := rxUdpData.AngRate_R;
feedback.wy := rxUdpData.AngRate_P;
feedback.wz := rxUdpData.AngRate_Y;
feedback.wx_t := rxUdpData.AngAcc_R;
feedback.wy_t := rxUdpData.AngAcc_P;
feedback.wz_t := rxUdpData.AngAcc_Y;
feedback.x_t := rxUdpData.VelMru_R;
feedback.y_t := rxUdpData.VelMru_P;
feedback.z_t := rxUdpData.VelMru_Y;
feedback.x_tt := rxUdpData.AccMru_R;
feedback.y_tt := rxUdpData.AccMru_P;
feedback.z_tt := rxUdpData.AccMru_Y;
END_METHOD

METHOD PRIVATE UpdateUDP : BOOL
VAR_INPUT
END_VAR
// Check for incoming UDP data
IF ipUdp <> 0 THEN
	ipUdp.CheckReceived();
END_IF

// TODO: Fix this ina  more elegant way
rxUdpData.mruOK := rxUdpDataBE.mruOK;
rxUdpData.dataLength := rxUdpDataBE.dataLength;
rxUdpData.token := rxUdpDataBE.token;
rxUdpData.checksum := rxUdpDataBE.checksum;

// Big to little endian real data conversion
rxUdpData.Temperature := BigToLittleEndian(rxUdpDataBE.Temperature);
rxUdpData.PosMru_D := BigToLittleEndian(rxUdpDataBE.PosMru_D);
rxUdpData.VelMru_D := BigToLittleEndian(rxUdpDataBE.VelMru_D);
rxUdpData.AccMru_D := BigToLittleEndian(rxUdpDataBE.AccMru_D);
rxUdpData.AngRate_D := BigToLittleEndian(rxUdpDataBE.AngRate_D);
rxUdpData.Roll := BigToLittleEndian(rxUdpDataBE.Roll);
rxUdpData.Pitch := BigToLittleEndian(rxUdpDataBE.Pitch);
rxUdpData.Yaw := BigToLittleEndian(rxUdpDataBE.Yaw);
rxUdpData.AngRate_R := BigToLittleEndian(rxUdpDataBE.AngRate_R);
rxUdpData.AngRate_P := BigToLittleEndian(rxUdpDataBE.AngRate_P);
rxUdpData.AngRate_Y := BigToLittleEndian(rxUdpDataBE.AngRate_Y);
rxUdpData.AngAcc_R := BigToLittleEndian(rxUdpDataBE.AngAcc_R);
rxUdpData.AngAcc_P := BigToLittleEndian(rxUdpDataBE.AngAcc_P);
rxUdpData.AngAcc_Y := BigToLittleEndian(rxUdpDataBE.AngAcc_Y);
rxUdpData.VelMru_R := BigToLittleEndian(rxUdpDataBE.VelMru_R);
rxUdpData.VelMru_P := BigToLittleEndian(rxUdpDataBE.VelMru_P);
rxUdpData.VelMru_Y := BigToLittleEndian(rxUdpDataBE.VelMru_Y);
rxUdpData.AccMru_R := BigToLittleEndian(rxUdpDataBE.AccMru_R);
rxUdpData.AccMru_P := BigToLittleEndian(rxUdpDataBE.AccMru_P);
rxUdpData.AccMru_Y := BigToLittleEndian(rxUdpDataBE.AccMru_Y);
END_METHOD

END_FUNCTION_BLOCK

// ---- POUs/Kinematics/EulerToBody.TcPOU
FUNCTION_BLOCK EulerToBody
VAR_INPUT
	roll : REAL := 0.0;
	pitch : REAL := 0.0;
	yaw : REAL := 0.0;
	
	roll_t : REAL := 0.0;
	pitch_t : REAL := 0.0;
	yaw_t : REAL := 0.0;
	
	roll_tt : REAL := 0.0;
	pitch_tt : REAL := 0.0;
	yaw_tt : REAL := 0.0;
END_VAR
VAR_OUTPUT
	wx : REAL := 0.0;
	wy : REAL := 0.0;
	wz : REAL := 0.0;
	
	wx_t : REAL := 0.0;
	wy_t : REAL := 0.0;
	wz_t : REAL := 0.0;
END_VAR
VAR
	phi : ARRAY [0..2] OF REAL;
	phi_t : ARRAY [0..2] OF REAL;
	phi_tt : ARRAY [0..2] OF REAL;
	
	w : ARRAY [0..2] OF REAL;
	w_t : ARRAY [0..2] OF REAL;
END_VAR

// Positions
phi[0] := roll;
phi[1] := pitch;
phi[2] := yaw;

// Velocities
phi_t[0] := roll_t;
phi_t[1] := pitch_t;
phi_t[2] := yaw_t;

// Accelerations
phi_tt[0] := roll_tt;
phi_tt[1] := pitch_tt;
phi_tt[2] := yaw_tt;

// Transform from phi_t to w
w[0] := phi_t[1]*SIN(phi[2]) + phi_t[0]*COS(phi[1])*COS(phi[2]);
w[1] := phi_t[1]*COS(phi[2]) - phi_t[0]*COS(phi[1])*SIN(phi[2]);
w[2] := phi_t[2] + phi_t[0]*SIN(phi[1]);

// Transform from phi_tt to w_t
w_t[0] := SIN(phi[2])*phi_tt[1] + COS(phi[2])*phi_t[1]*phi_t[2] + COS(phi[1])*COS(phi[2])*phi_tt[0] - COS(phi[2])*SIN(phi[1])*phi_t[0]*phi_t[1] - COS(phi[1])*SIN(phi[2])*phi_t[0]*phi_t[2];
w_t[1] := COS(phi[2])*phi_tt[1] - SIN(phi[2])*phi_t[1]*phi_t[2] - COS(phi[1])*SIN(phi[2])*phi_tt[0] - COS(phi[1])*COS(phi[2])*phi_t[0]*phi_t[2] + SIN(phi[1])*SIN(phi[2])*phi_t[0]*phi_t[1];
w_t[2] := SIN(phi[1])*phi_tt[0] + phi_tt[2] + COS(phi[1])*phi_t[0]*phi_t[1];

// Rotational velocites in body coordinates
wx := w[0];
wy := w[1];
wz := w[2];

// Rotational accelerations in body coordinates
wx_t := w_t[0];
wy_t := w_t[1];
wz_t := w_t[2];

END_FUNCTION_BLOCK

// ---- POUs/Kinematics/StewartTransform.TcPOU
PROGRAM StewartTransform
VAR
END_VAR

METHOD PRIVATE xyz2zyx : ARRAY [0..2] OF REAL
VAR_INPUT
	phi : ARRAY [0..2] OF REAL;
END_VAR

VAR
	t1: REAL;
	t2: REAL;
	t3: REAL;
	t4: REAL;
	t5: REAL;
	t6: REAL;
	t7: REAL;
	t8: REAL;
END_VAR
// Maple optimized code
t1 := COS(phi[0]);
t2 := SIN(phi[1]);
t3 := SIN(phi[2]);
t4 := SIN(phi[0]);
t5 := COS(phi[2]);
t6 := t1 * t3;
t7 := t4 * t5;
t8 := COS(phi[1]);

xyz2zyx[0] := ATAN((t6 * t2 + t7)/(t1 * t8));
xyz2zyx[1] := -ASIN(-t1 * t2 * t5 + t3 * t4);
xyz2zyx[2] := ATAN((t7 * t2 + t6)/(t5 * t8));
END_METHOD

METHOD PRIVATE zyx2xyz : ARRAY [0..2] OF REAL
VAR_INPUT
	phi : ARRAY [0..2] OF REAL;
END_VAR

VAR
	t1: REAL;
	t2: REAL;
	t3: REAL;
	t4: REAL;
	t5: REAL;
	t6: REAL;
	t7: REAL;
	t8: REAL;
END_VAR
// Maple optimized code
t1 := SIN(phi[0]);
t2 := COS(phi[2]);
t3 := COS(phi[0]);
t4 := SIN(phi[1]);
t5 := SIN(phi[2]);
t6 := t3 * t5;
t7 := t1 * t2;
t8 := COS(phi[1]);

zyx2xyz[0] := ATAN((-t6 * t4 + t7)/(t3 * t8));
zyx2xyz[1] := ASIN(t3 * t4 * t2 + t1 * t5);
zyx2xyz[2] := ATAN((-t7 * t4 + t6)/( t2 * t8));
END_METHOD

END_PROGRAM

// ---- POUs/Ship Simulation/StocWave.TcPOU
FUNCTION StocWave : REAL
VAR_INPUT
	Tp			: REAL := 20.0;
	Hs			: REAL := 0.20;
	t			: REAL := 0.0;
	mode		: INT := 0;
END_VAR
VAR
	// Random phases
	phi_0		: ARRAY [1..25] OF REAL := [4.761022,4.669239,2.464435,4.118489,1.075598,4.436218,0.200012,1.739958,0.290103,0.610297,5.173938,4.365737,1.992395,5.970421,0.216431,2.756712,2.397402,4.809884,4.996388,1.174155,3.077280,2.799701,4.060904,4.457071,4.741836];
	phi_1		: ARRAY [1..25] OF REAL := [1.734317,4.270698,4.116102,1.021720,0.747684,3.131314,6.030249,2.138707,3.677346,1.406252,4.720350,1.602810,3.179022,4.392429,5.597710,6.027406,3.438257,0.871003,0.938042,1.617972,5.282382,1.597702,5.116302,1.530113,5.838736];
	phi_2		: ARRAY [1..25] OF REAL := [2.199013,1.235244,1.577606,3.870723,2.973762,2.209542,5.220250,3.677323,3.454015,5.762898,1.795980,4.757629,4.735820,2.390412,3.567729,0.476607,0.338979,3.335099,4.895652,5.868562,0.816225,3.574024,2.949268,0.074783,2.118204];
	phi_3		: ARRAY [1..25] OF REAL := [1.019021,4.990637,1.955422,3.320872,1.040802,3.782364,1.652297,4.109700,4.330462,4.700775,2.830836,0.526665,1.438705,5.738668,0.957419,5.188761,3.382505,6.258899,0.491191,2.781430,0.670119,6.043784,0.029118,4.868906,5.135268];
	
	i 			: INT;
	dw			: REAL;
	w			: REAL;
	Sx			: REAL;
	pi			: REAL := 3.141592653589793;
	An			: REAL := 0.0;
	xn			: REAL := 0.0;
	x			: REAL := 0.0;
END_VAR



dw	:= 1.0/25.0;
x := 0.0;
FOR i := 1 TO 25 BY 1 DO
	// Frequency componen i
	w := dw*INT_TO_REAL(i);
	
	// Calculate the wave spectrum
	Sx := LREAL_TO_REAL(5*EXPT(pi,4)*EXPT(Hs,2)/(EXPT(Tp,4)*EXPT(w,5))*EXP(-20*EXPT(pi,4)/(EXPT(Tp,4)*EXPT(w,4))));
	
	// Wave component i
	An := SQRT(2*Sx*dw);
	
	CASE mode OF
	0 :
		xn := An*SIN(w*t-phi_0[i]);
	1 :
		xn := An*SIN(w*t-phi_1[i]);
	2 :
		xn := An*SIN(w*t-phi_2[i]);
	3 :
		xn := An*SIN(w*t-phi_3[i]);
	ELSE
		xn := 0.0;
	END_CASE;
	
	// Sum up output wave signal
	x := x + xn;
END_FOR;

// Return the wave amplitude
StocWave := x;

END_FUNCTION

// ---- POUs/UdpFBs/FB_UdpServer.TcPOU
{attribute 'c++_compatible'}
FUNCTION_BLOCK FB_UdpServer IMPLEMENTS ITcIoUdpProtocolRecv
VAR_INPUT
	
END_VAR
VAR_OUTPUT
	
END_VAR
VAR
	{attribute 'TcInitSymbol'}
	oid					: OTCID;
	ipUdp 				: ITcIoUdpProtocol;
	nSendPackets		: UDINT := 0;
	nReceivedPackets	: UDINT := 0;
	
	// Values are initilized in FB_init
	nLocalPort			: UINT;
	nDataSend 			: UDINT;
	pDataSend			: PVOID;
	nDataRecv			: UDINT;
	pDataRecv			: PVOID;
END_VAR

IF ipUdp <> 0 THEN
	// If data is recieved, receive data method is called
	ipUdp.CheckReceived();
END_IF

METHOD FB_exit : BOOL
VAR_INPUT
	bInCopyCode : BOOL; // if TRUE, the exit method is called for exiting an instance that is copied afterwards (online change).
END_VAR
IF (NOT bInCopyCode AND ipUdp <> 0) THEN //Shutdown
	ipUdp.UnregisterReceiver(nLocalPort);
	FW_SafeRelease(ADR(ipUdp));
	FB_exit := TRUE;
ELSE
	FB_exit := FALSE;
END_IF
END_METHOD

METHOD FB_init : BOOL
VAR_INPUT
	bInitRetains			: BOOL; 	// if TRUE, the retain variables are initialized (warm start / cold start)
	bInCopyCode				: BOOL;  	// if TRUE, the instance afterwards gets moved into the copy code (online change)
	nLocalPortInit			: UINT;
	nDataSendInit 			: UDINT;
	pDataSendInit			: PVOID;
	nDataRecvInit 			: UDINT;
	pDataRecvInit			: PVOID;
END_VAR
VAR
	ipSrv: ITComObjectServer;
	hr : HRESULT;
END_VAR
// Initilize the port
nLocalPort 		:= nLocalPortInit;

nDataSend 		:= nDataSendInit;
pDataSend 		:= pDataSendInit;

nDataRecv	 	:= nDataRecvInit;
pDataRecv	 	:= pDataRecvInit;

IF NOT bInCopyCode THEN // no online change
	IF ipUdp = 0 THEN
	    hr := FW_ObjMgr_GetObjectInstance(oid:=oid, iid:=TC_GLOBAL_IID_LIST.IID_ITcIoUdpProtocol, pipUnk:=ADR(ipUdp) );
		
		IF ( SUCCEEDED(hr) AND ipUdp.RegisterReceiver(nLocalPort, THIS^) = 0 ) THEN //open local port
			FB_init := TRUE;
		ELSE
			FB_init := FALSE;			
			FW_SafeRelease(ADR(ipUdp));
		END_IF				
	END_IF
END_IF
END_METHOD

METHOD FB_reinit : BOOL
VAR_INPUT
END_VAR
IF (ipUdp <> 0) THEN 
	ipUdp.RegisterReceiver(nLocalPort, THIS^);
END_IF
END_METHOD

{attribute 'object_name' := 'ReceiveData'}
{attribute 'c++_compatible'}
{attribute 'signature_flag' := '33554688'}
{attribute 'pack_mode' := '4'}
{attribute 'show'}
{attribute 'minimal_input_size' := '4'}
METHOD ReceiveData : HRESULT
VAR_INPUT
	ipAddr			: UDINT;
	udpDestPort		: UINT;
	udpSrcPort		: UINT;
	nData			: UDINT;
	pData			: PVOID;
	pVlan			: POINTER TO ETYPE_VLAN_HEADER := 0;
END_VAR

VAR
	
END_VAR
// Count number of recieved UDP packets
nReceivedPackets := nReceivedPackets + 1;

// Send and receive data if the received data size is correct
IF (nData = nDataRecv) THEN
	// Receive data
	MEMCPY(pDataRecv, pData, nDataRecv);
	
	// Send data
	ipUdp.SendData(ipAddr, udpSrcPort, udpDestPort, nDataSend, pDataSend, TRUE, 0);
	nSendPackets := nSendPackets + 1;
ELSE;
	// Return the same data as recevied
	ipUdp.SendData(ipAddr, udpSrcPort, udpDestPort, nData, pData, TRUE, 0);
END_IF
END_METHOD

{attribute 'object_name' := 'TcAddRef'}
{attribute 'c++_compatible'}
{attribute 'signature_flag' := '33554688'}
{attribute 'pack_mode' := '4'}
{attribute 'show'}
{attribute 'minimal_input_size' := '4'}
METHOD TcAddRef : UDINT
END_METHOD

{attribute 'object_name' := 'TcQueryInterface'}
{attribute 'c++_compatible'}
{attribute 'signature_flag' := '33554688'}
{attribute 'pack_mode' := '4'}
{attribute 'show'}
{attribute 'minimal_input_size' := '4'}
METHOD TcQueryInterface : HRESULT
VAR_INPUT
	iid	: REFERENCE TO IID;
	pipItf	: POINTER TO PVOID;
END_VAR
END_METHOD

{attribute 'object_name' := 'TcRelease'}
{attribute 'c++_compatible'}
{attribute 'signature_flag' := '33554688'}
{attribute 'pack_mode' := '4'}
{attribute 'show'}
{attribute 'minimal_input_size' := '4'}
METHOD TcRelease : UDINT
END_METHOD

END_FUNCTION_BLOCK

// ---- GlobalTextList.TcGTLO
TEXTLIST GlobalTextList
  26 = '%5.2f'
  25 = '%5.f'
  24 = '%d'
  5 = '%f'
  6 = '%i'
  46 = '%if'
  57 = 'Activate Camera'
  37 = 'Cal Pitch'
  33 = 'Cal X'
  34 = 'Cal Y'
  36 = 'Cal Yaw'
  35 = 'Cal Z'
  39 = 'Comau Robot'
  28 = 'COMAU Smart 5'
  56 = 'Deactivate Camera'
  15 = 'E-Motion 1500'
  14 = 'E-Motion 8000'
  0 = 'EM1500'
  49 = 'filt_phi'
  45 = 'filt_x'
  47 = 'filt_y'
  48 = 'filt_z'
  30 = 'High Speed'
  31 = 'Low Speed'
  42 = 'omega'
  12 = 'Pitch'
  50 = 'q'
  16 = 'q1'
  17 = 'q2'
  18 = 'q3'
  19 = 'q4'
  20 = 'q5'
  21 = 'q6'
  54 = 'qStd'
  52 = 'qVar'
  51 = 'r'
  29 = 'Reset all inputs to default'
  10 = 'Reset all inputs to zero'
  4 = 'Reset and Settled'
  11 = 'Roll'
  55 = 'rStd'
  53 = 'rVar'
  3 = 'To Engaged'
  41 = 'To Engaged - Fast'
  40 = 'To Engaged - Slow'
  44 = 'To Engaged/Freeze'
  32 = 'To Manual Engaged'
  2 = 'To Neutral'
  1 = 'To Settled'
  38 = 'To Settled\t'
  43 = 'To Settled and Reset'
  58 = 'ux'
  59 = 'uy'
  60 = 'uz'
  7 = 'X'
  22 = 'x'
  8 = 'Y'
  27 = 'y'
  13 = 'Yaw'
  9 = 'Z'
  23 = 'z'
END_TEXTLIST
